FUNCTION_BLOCK FB_Restoration_SFC EXTENDS FB_Object_Template_ST
VAR_INPUT
END_VAR
VAR_OUTPUT
END_VAR
VAR
END_VAR

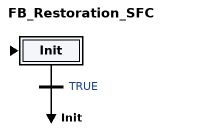
INITIAL_STEP Init:
END_STEP
TRANSITION FROM Init TO Init
    := TRUE;
END_TRANSITION

END_FUNCTION_BLOCK

(* stored: Version 1.1.0.1, ProductVersion 3.1.4024.6
   POU FB_Restoration_SFC: Id {1d0fac57-71a8-4305-a9f7-ceeeac47bd4e}, SpecialFunc None *)
